(* CoDeSys 2.3.9.50 project: me308servo.pro *)
(* Libraries: TcBase.lib 14.5.09 12:14:08, TcSystem.lib 7.6.16 11:01:22, TcMc2Drive.lib 9.10.17 15:27:28, TcBaseMath.lib 27.7.04 12:07:56, TcMath.lib 23.9.04 15:15:30, TcMC2.lib 13.9.17 10:18:38, TcUtilities.lib 3.2.16 16:08:58, TcEtherCAT.lib*30.11.16 19:52:18, TcTestAndSet.lib 23.2.09 12:50:08, TcDrive.lib 25.1.17 09:42:28, STANDARD.LIB 5.6.98 12:03:02, SysLibVisu.lib 7.7.04 18:17:22, SysLibTargetVisu.lib 16.6.08 16:24:26 *)

(* Task configuration *)
TASK Standard (PRIORITY := 0, INTERVAL := T#10ms);
	MAIN
END_TASK
TASK VISU_TASK (PRIORITY := 3, INTERVAL := T#200ms);
	MAINTARGETVISU_PAINT_CODE
END_TASK
TASK VISU_INPUT_TASK (PRIORITY := 2, INTERVAL := T#50ms);
	MAINTARGETVISU_INPUT_CODE
END_TASK

(* Global variable list: TwinCAT_Configuration *)
(* Generated automatically by TwinCAT - (read only) *)
VAR_CONFIG
	MAIN.First_Axis.PlcToNc AT %QB0 : PLCTONC_AXIS_REF;	(*  ~ {LinkedWith:TINC^NC-Task 1 SAF^Axes^Axis 1^Inputs^Axis 1_FromPlc} *)
	MAIN.First_Axis.NcToPlc AT %IB0 : NCTOPLC_AXIS_REF;	(*  ~ {LinkedWith:TINC^NC-Task 1 SAF^Axes^Axis 1^Outputs^Axis 1_ToPlc} *)
	MAIN.Second_Axis.PlcToNc AT %QB128 : PLCTONC_AXIS_REF;
	MAIN.Second_Axis.NcToPlc AT %IB128 : NCTOPLC_AXIS_REF;
END_VAR

(* POU MAIN, ST *)
PROGRAM MAIN
VAR
	First_Axis: AXIS_REF;
	First_Axis_Power:MC_Power;
	First_Axis_Reset:MC_Reset;
	First_Axis_Jog:MC_Jog;
	First_Axis_SoEReset:FB_SoEReset;

	First_Axis_enable_command:BOOL;
	First_Axis_status_flag:BOOL;

	First_Axis_Move_Absolute:MC_MoveAbsolute;

	First_Axis_Move_AbsoluteExecute:BOOL;
	First_Axis_Move_AbsolutePosition:LREAL;
	First_Axis_Move_AbsoluteVelocity:LREAL;
	First_Axis_Move_AbsoluteAcceleration:LREAL;
	First_Axis_Move_AbsoluteDeceleration:LREAL;
	First_Axis_Move_AbsoluteJerk:LREAL;

	First_Axis_Move_AbsoluteDone:BOOL;

	First_Axis_Actual_Position:LREAL;

	h001_firstaxisexe_execute_button_pressed:BOOL;
	h001_firstaxisexe_execute_button_pressed_rising_edge:R_TRIG;
	h001_firstaxisexe_done_rising_edge:R_TRIG;


	Second_Axis:AXIS_REF;
	Second_Axis_Power:MC_Power;
	Second_Axis_Reset:MC_Reset;
	Second_Axis_Jog:MC_Jog;
	Second_Axis_SoEReset:FB_SoEReset;
END_VAR
First_Axis_Power
	(Enable:=First_Axis_enable_command,
	Enable_Positive:=First_Axis_enable_command,
	Enable_Negative:=First_Axis_enable_command,
	Override:=100,
	Axis:=First_Axis);
First_Axis_status_flag:=First_Axis_Power.Status;
First_Axis_Move_Absolute
	(Execute:=First_Axis_Move_AbsoluteExecute,
	Position:=First_Axis_Move_AbsolutePosition,
	Velocity:=First_Axis_Move_AbsoluteVelocity,
	Acceleration:=First_Axis_Move_AbsoluteAcceleration,
	Deceleration:=First_Axis_Move_AbsoluteDeceleration,
	Jerk:=First_Axis_Move_AbsoluteJerk,
	Axis:=First_Axis);

First_Axis_Move_AbsoluteDone:= First_Axis_Move_Absolute.Done;
First_Axis_Actual_position:=First_Axis.NcToPlc.ActPos;

First_Axis_Move_AbsoluteVelocity:=100;
First_Axis_Move_AbsoluteAcceleration:=200;
First_Axis_Move_AbsoluteDeceleration:=200;
First_Axis_Move_AbsoluteJerk:=0;

h001_first_axis_execute_handling();
END_PROGRAM
ACTION h001_first_axis_execute_handling:
h001_firstaxisexe_execute_button_pressed_rising_edge
	(CLK:=h001_firstaxisexe_execute_button_pressed);

IF h001_firstaxisexe_execute_button_pressed_rising_edge.Q THEN
	First_Axis_Move_AbsoluteExecute:=TRUE;
END_IF

h001_firstaxisexe_done_rising_edge
	(CLK:=First_Axis_Move_AbsoluteDone AND NOT
		h001_firstaxisexe_execute_button_pressed);

IF h001_firstaxisexe_done_rising_edge.Q THEN
	First_Axis_Move_AbsoluteExecute:=FALSE;
END_IF
END_ACTION

(* Visualisation V001_SERVO_PAGE
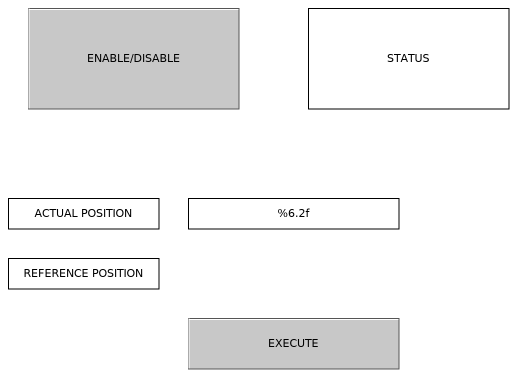
rectangle at (340,70)-(541,171): text "STATUS"; alarm colour if MAIN.First_Axis_status_flag
button at (60,70)-(271,171): text "ENABLE/DISABLE"; toggles MAIN.First_Axis_enable_command
rectangle at (220,260)-(431,291): text "%6.2f"; shows MAIN.First_Axis_Actual_Position
rectangle at (40,260)-(191,291): text "ACTUAL POSITION"
rectangle at (40,320)-(191,351): text "REFERENCE POSITION"
button at (220,380)-(431,431): text "EXECUTE"; taps MAIN.First_Axis_Move_AbsoluteExecute
1 elements of other kinds (tables, trends, ...) not read
*)
